FUNCTION_BLOCK ST80c
VAR
	_promenlivaNova		: BOOL;
	_ivana : INT;
	_test : BOOL;
END_VAR

METHOD _test : BOOL
VAR_INPUT
END_VAR
IF _test THEN 
	_ivana:= 5;
ELSE 
_ivana:= 3; 
END_IF
END_METHOD

END_FUNCTION_BLOCK

(* stored: Version 1.1.0.1, ProductVersion 3.1.4024.12
   POU ST80c: Id {6511e522-115d-43cb-a766-5883ce869da5}, SpecialFunc None
   Method _test: Id {4745666f-855a-404a-9b5b-260c04e7b323} *)
